Staubli VAL3: Rob6x.pjx

--- Rob6x.pjx ---
Parameters version=s7.9.1 stackSize=5000 millimeterUnit=true
Program file=AsynchStop.pgx
Program file=BytesToS16.pgx
Program file=Calibrate.pgx
Program file=CheckLimits.pgx
Program file=CheckStatus.pgx
Program file=Com.pgx
Program file=COM_SERIAL.pgx
Program file=Command.pgx
Program file=crc16.pgx
Program file=DeletePoint.pgx
Program file=Energize.pgx
Program file=FloatToBytes.pgx
Program file=GetAppVersion.pgx
Program file=GetCurrentPos.pgx
Program file=GetFirmVersion.pgx
Program file=GetJointPos.pgx
Program file=GetLimits.pgx
Program file=GetSerialNumber.pgx
Program file=GetSNCtrl.pgx
Program file=GetToolParam6x.pgx
Program file=GotoPoint.pgx
Program file=GotoPosition.pgx
Program file=Init.pgx
Program file=InitRobot.pgx
Program file=Input.pgx
Program file=isInLimits.pgx
Program file=KillAlltasks.pgx
Program file=MemPointPos.pgx
Program file=Motion.pgx
Program file=Move.pgx
Program file=MoveJoint.pgx
Program file=MoveJointTo.pgx
Program file=Output.pgx
Program file=SetAccel.pgx
Program file=SetLimits.pgx
Program file=SetSpeed.pgx
Program file=SetTool.pgx
Program file=SetToolParam.pgx
Program file=SetToolParam6x.pgx
Program file=start.pgx
Program file=stop.pgx
Program file=StopLimits.pgx
Program file=taskRecord.pgx
Program file=test.pgx
Program file=Valve.pgx
Data file=Rob6x.dtx

--- CheckLimits.pgx ---
program CheckLimits()
  local pointRx pt
  local bool curErr_Z
  local bool err_x
  local bool err_y
  local bool curErr_Y
  local bool err_z
  local num hysteresis
  local bool curErr_X
  local bool inLimits
  local num hysteresisZmin
begin
//*******************************************************************************
//*   ______
//*  / _____) /|
//* | |      / /
//* | | /\  / /
//* | | \ \/ /  _      Copyright (c) KEOLABS, 2016
//* | |  \__/  | |        http://www.keolabs.com
//* | |________| |
//*  \__________/
//*
//********************************************************************************
//*@file          : CheckLimits
//*@author        : Yves Ragot
//*@version       : $Id: CheckLimits.pgx 1645 2017-01-24 08:09:09Z yves $
//*@brief         : Check the if the current mouvement is in the limits
//*
//*******************************************************************************/

  // hysteresis in mm
  hysteresis = 70
  hysteresisZmin = 10

  do

      // get current position
      pt = here(tCurrentTool, fCurrentFrame)

      // round values before comparing with limits (integer values)
      pt.trsf.x = round(pt.trsf.x * 10) / 10
      pt.trsf.y = round(pt.trsf.y * 10) / 10
      pt.trsf.z = round(pt.trsf.z * 10) / 10

      // check first non fatal X limits
      if ((pt.trsf.x < CurLimitsTable["Xmin"]) or (pt.trsf.x > CurLimitsTable["Xmax"]))
          if (!curErr_X)
              call StopLimits()
          endIf
      else
          curErr_X = false
      endIf

      if ((pt.trsf.x >= CurLimitsTable["Xmin"] - hysteresis) and (pt.trsf.x <= CurLimitsTable["Xmax"] + hysteresis))
          curErr_X = true
      else
          call StopLimits()
      endIf

      // check first non fatal Y limits
      if ((pt.trsf.y < CurLimitsTable["Ymin"]) or (pt.trsf.y > CurLimitsTable["Ymax"]))
          if (!curErr_Y)
              call StopLimits()
          endIf
      else
          curErr_Y = false
      endIf

      if ((pt.trsf.y >= CurLimitsTable["Ymin"] - hysteresis) and (pt.trsf.y <= CurLimitsTable["Ymax"] + hysteresis))
          curErr_Y = true
      else
          call StopLimits()
      endIf

      // check first non fatal Z limits
      if ((pt.trsf.z < CurLimitsTable["Zmin"]) or (pt.trsf.z > CurLimitsTable["Zmax"]))
          if (!curErr_Z)
              call StopLimits()
          endIf
      else
          curErr_Z = false
      endIf

      if ((pt.trsf.z >= CurLimitsTable["Zmin"] - hysteresisZmin) and (pt.trsf.z <= CurLimitsTable["Zmax"] + hysteresis))
          curErr_Z = true
      else
          call StopLimits()
      endIf

     delay(0)

  until false

end

--- CheckStatus.pgx ---
program CheckStatus()
  local num esState
  local num status_err
  local num com_err
  local num limits_err
  local num motion_err
  local num newErrorCode
begin
//*******************************************************************************
//*   ______
//*  / _____) /|
//* | |      / /
//* | | /\  / /
//* | | \ \/ /  _      Copyright (c) KEOLABS, 2016
//* | |  \__/  | |        http://www.keolabs.com
//* | |________| |
//*  \__________/
//*
//********************************************************************************
//*@file          : CheckStatus
//*@author        : Yves Ragot
//*@version       : $Id: CheckStatus.pgx 1365 2016-11-18 16:00:54Z yves $
//*@brief         : Check robot status (busy, runing, error ?)
//*
//*******************************************************************************/

  do

      //== get task errors ==
      com_err = taskStatus("COM")
      limits_err = taskStatus("CheckLimits")
      status_err = taskStatus("CheckStatus")
      motion_err = taskStatus("Motion")

      // update LastErrorCode (taskStatus: 0 = suspended, 1 = running, -1 = dead
      if ((com_err != 0) and (com_err != 1))
          newErrorCode = com_err
      elseIf (motion_err > 1)
          newErrorCode = motion_err
      elseIf ((limits_err != 0) and (limits_err != 1))
          newErrorCode = limits_err
      elseIf ((status_err != 0) and (status_err != 1))
          newErrorCode = status_err
      else
          newErrorCode = 0
      endIf

      //== GeneralStatus
      // emergency stop ?
      esState = esStatus()
      if (esState != 0)
          call AsynchStop()
          GeneralStatus = 105
          LastErrorCode = 0

      // mouvement error ?
      elseIf (GeneralStatus == 0)

        switch (newErrorCode)

          // mouvement
          case 81, 150, 153, 154
            GeneralStatus = 100
          break

          // parameter
          case 70, 100, 101, 102, 103, 104, 160, 161, 165
            GeneralStatus = 101
          break

          // system
          case -1, 40, 41, 60, 61, 90, 125, 250
            GeneralStatus = 102
          break

          // soft
          case 10, 11, 20, 21, 29, 30, 31, 32, 80, 82, 105, 106, 122, 123, 124, 162, 163, 164
            GeneralStatus = 103
          break

          default
          break

        endSwitch

        if (newErrorCode != 0)
            LastErrorCode = newErrorCode
        endIf

    endIf

      // kill motion task if fault
    //    if ((GeneralStatus > 1) and (LastErrorCode != 0) and ((LastErrorCode == motion_err) or (LastErrorCode == 153)))
    if ((MoveRunning and (GeneralStatus > 1) and ((LastErrorCode == motion_err) or (LastErrorCode == 153))))
        call AsynchStop()
        setMutex(MotionTaskMutex)
        if taskStatus("Motion") != -1
            taskKill("Motion")
            wait(taskStatus("Motion") == -1)
            ExecuteMotion = false
        endIf
        MotionTaskMutex = false
    endIf

    // check movement running
    if (GeneralStatus == 1)
        // is mouvement always running ?
        if (isSettled() and isEmpty())
            GeneralStatus = 0
            MoveRunning = false
        endIf
    endIf

   delay(0)

  until false

end

--- Com.pgx ---
program COM()
  local num nbBuffer
  local num nbSent
  local num dataIn[50]
  local num dataOut[32]
  local num crc_l
  local num crc_h
  local num ret
  local num lenDataIn
  local num lenDataOut
  local num answer
  local string stringAnswer
  local num i
  local num j
  local num arrayAnswer[6]
  local num buffer[64]
  local num l_nIndex
  local num cpt
  local num nbBufTcp
  local num bufferTCP[64]
begin
//*******************************************************************************
//*   ______
//*  / _____) /|
//* | |      / /
//* | | /\  / /
//* | | \ \/ /  _      Copyright (c) KEOLABS, 2016
//* | |  \__/  | |        http://www.keolabs.com
//* | |________| |
//*  \__________/
//*
//********************************************************************************
//*@file          : COM
//*@author        : Yves Ragot
//*@version       : $Id: Com.pgx 1608 2017-01-13 10:03:43Z yves $
//*@brief         : PC socket communication management
//*
//*******************************************************************************/

  //== configuration socket ==
  // 1 seul client
  ret = sioCtrl(siTcpServer, "clients", 1)

  // timeout = 10ms
  ret = sioCtrl(siTcpServer, "timeout", 0.01)

  // buffers length
  lenDataIn = 32
  lenDataOut = 32

  NbCharReceived = 0
  ModeSerial = false

  // auto detection com port with first frame
  do
    nbBufTcp = sioGet(siTcpServer, bufferTCP)
  until ((NbBufSerial > 0) or (nbBufTcp > 0))

  // serial detection done by COM_SERIAL task
  if (NbBufSerial > 0)
      nbBuffer = NbBufSerial
      ModeSerial = true
  endIf
  if (nbBufTcp > 0)
      nbBuffer = nbBufTcp
      ModeSerial = false
  endIf

  if (nbBuffer > lenDataIn)
      nbBuffer = lenDataIn
  endIf

  if (ModeSerial)
      for l_nIndex = 0 to nbBuffer
          dataIn[NbCharReceived + l_nIndex] = BufferSerial[l_nIndex]
      endFor
  else
      for l_nIndex = 0 to nbBuffer
          dataIn[NbCharReceived + l_nIndex] = bufferTCP[l_nIndex]
      endFor
  endIf

  NbCharReceived = NbCharReceived + nbBuffer

  // main loop
  do

      cpt = 0

      do
          if (ModeSerial)
              nbBuffer = sioGet(siSerial1, buffer)
          else
              nbBuffer = sioGet(siTcpServer, buffer)
          endIf

          if (nbBuffer > 0)
              if (nbBuffer > lenDataIn)
                  nbBuffer = lenDataIn
              endIf
              if (NbCharReceived + nbBuffer > lenDataIn)
                  NbCharReceived = lenDataIn
              else

                  for l_nIndex = 0 to nbBuffer
                      dataIn[NbCharReceived + l_nIndex] = buffer[l_nIndex]
                  endFor
                  NbCharReceived = NbCharReceived + nbBuffer
                  cpt = cpt + 1
              endIf

          endIf

      // loop on charactere until all frame or 1s timeout
      until (NbCharReceived == lenDataIn) or cpt > 100

    if (NbCharReceived == lenDataIn)

      // check CRC
      call crc16(lenDataIn - 2, crc_h, crc_l, dataIn)

      if ((dataIn[lenDataIn - 2] != crc_h) or (dataIn[lenDataIn - 1] != crc_l))
          FrameReceiveNOK = FrameReceiveNOK + 1
      else
          FrameReceiveOK = FrameReceiveOK + 1

        //== command treatment ==
        setMutex(MotionTaskMutex)
        if  (taskStatus("Motion") == -1)
            taskCreate "Motion", 100, Motion()
        endIf

        // be sure that the task is running
        wait(taskStatus("Motion") == 1)
        MotionTaskMutex = false

        call Command(ret, dataIn, answer, stringAnswer, arrayAnswer)

        //== prepare response ==

        // command number
        dataOut[0] = dataIn[0]

        // frame number
        dataOut[1] = dataIn[1]

        // last error code
        dataOut[2] = LastErrorCode

        // status
        dataOut[3] = GeneralStatus

        // check response type
        switch (dataIn[0])

          // string
          case 10, 11, 13, 15
              for i = 0 to len(stringAnswer) - 1
                  dataOut[4 + i] = asc(stringAnswer, i)
              endFor
              for j = i to 24
                  dataOut[4 + j] = 0
              endFor
          break

          // numerical or nothing
          default
              // if not limits or ToolParam
              if ((dataIn[0] != 6) and (dataIn[0] != 16))
                  // current Cartesian position
                  call GetCurrentPos(arrayAnswer)
              endIf

              call FloatToBytes(arrayAnswer[0], dataOut[4], dataOut[5])
              call FloatToBytes(arrayAnswer[1], dataOut[6], dataOut[7])
              call FloatToBytes(arrayAnswer[2], dataOut[8], dataOut[9])
              call FloatToBytes(arrayAnswer[3], dataOut[10], dataOut[11])
              call FloatToBytes(arrayAnswer[4], dataOut[12], dataOut[13])
              call FloatToBytes(arrayAnswer[5], dataOut[14], dataOut[15])

              // current Joint position
              call GetJointPos(arrayAnswer)
              call FloatToBytes(arrayAnswer[0], dataOut[16], dataOut[17])
              call FloatToBytes(arrayAnswer[1], dataOut[18], dataOut[19])
              call FloatToBytes(arrayAnswer[2], dataOut[20], dataOut[21])
              call FloatToBytes(arrayAnswer[3], dataOut[22], dataOut[23])
              call FloatToBytes(arrayAnswer[4], dataOut[24], dataOut[25])
              call FloatToBytes(arrayAnswer[5], dataOut[26], dataOut[27])

              // command response (GetAccel/GetSpeed/GetToolParam or not)
              if (dataIn[0] == 3) or (dataIn[0] == 4) or (dataIn[0] == 5)
                  call FloatToBytes(answer, dataOut[28], dataOut[29])
              else
                  dataOut[28] = answer
              endIf
            break

        endSwitch

          // compute CRC
          call crc16(lenDataOut - 2, crc_h, crc_l, dataOut)
          dataOut[lenDataOut - 2] = crc_h
          dataOut[lenDataOut - 1] = crc_l

        // send response
        if (ModeSerial)
            nbSent = sioSet(siSerial1, dataOut)
        else
            nbSent = sioSet(siTcpServer, dataOut)
        endIf

        if (nbSent != lenDataOut)
            // TODO error
        endIf

        //if ((dataIn[30] != crc_h) or (dataIn[31] != crc_l))
      endIf

        //if (nbReceived == lenDataIn)
      elseIf (NbCharReceived > 0)
          FrameReceiveNOK = FrameReceiveNOK + 1
      endIf

      NbCharReceived = 0

      delay(0)

  until(bExit)

end

--- DeletePoint.pgx ---
program DeletePoint(num& bufferIn[])
  local string pointName
  local num i
begin
  //*******************************************************************************
  //*   ______
  //*  / _____) /|
  //* | |      / /
  //* | | /\  / /
  //* | | \ \/ /  _      Copyright (c) KEOLABS, 2016
  //* | |  \__/  | |        http://www.keolabs.com
  //* | |________| |
  //*  \__________/
  //*
  //********************************************************************************
  //*@file          : DeletePoint
  //*@author        : Yves Ragot
  //*@version       : $Id: DeletePoint.pgx 1198 2016-10-07 06:48:14Z yves $
  //*@brief         : Forget a memorized position point
  //*
  //*******************************************************************************/

  pointName = ""

  // get the name of the point
  for i = 0 to 9
      pointName = pointName + chr(bufferIn[17 + i])
  endFor

  if (len(pointName)) > 0

      // delete the point from the collection
      if (isDefined(pPointsTable[pointName]) == true)
          delete(pPointsTable[pointName])
      else
          GeneralStatus = 101
          LastErrorCode = 0
      endIf

  else
      GeneralStatus = 101
      LastErrorCode = 0
  endIf

end

--- GetAppVersion.pgx ---
program GetAppVersion(string& answer)
begin
//*******************************************************************************
//*   ______
//*  / _____) /|
//* | |      / /
//* | | /\  / /
//* | | \ \/ /  _      Copyright (c) KEOLABS, 2016
//* | |  \__/  | |        http://www.keolabs.com
//* | |________| |
//*  \__________/
//*
//********************************************************************************
//*@file          : GetAppVersion
//*@author        : Yves Ragot
//*@version       : $Id: GetAppVersion.pgx 1645 2017-01-24 08:09:09Z yves $
//*@brief         : Get firmware version (application version)
//*******************************************************************************/

  answer = "v1.1 jan 23 2017"

end

--- GetJointPos.pgx ---
program GetJointPos(num& posArray[])
  local jointRx jt
begin
  //*******************************************************************************
  //*   ______
  //*  / _____) /|
  //* | |      / /
  //* | | /\  / /
  //* | | \ \/ /  _      Copyright (c) KEOLABS, 2016
  //* | |  \__/  | |        http://www.keolabs.com
  //* | |________| |
  //*  \__________/
  //*
  //********************************************************************************
  //*@file          : GetJointPos
  //*@author        : Yves Ragot
  //*@version       : $Id: GetJointPos.pgx 1198 2016-10-07 06:48:14Z yves $
  //*@brief         : Get current joint position
  //*
  //*******************************************************************************/

  // get joint position and converts to 1/10 mm
  jt = herej()
  posArray[0] = jt.j1 * 10
  posArray[1] = jt.j2 * 10
  posArray[2] = jt.j3 * 10
  posArray[3] = jt.j4 * 10
  posArray[4] = jt.j5 * 10
  posArray[5] = jt.j6 * 10

end

--- GetLimits.pgx ---
program GetLimits(num& limits[])
begin
  //*******************************************************************************
  //*   ______
  //*  / _____) /|
  //* | |      / /
  //* | | /\  / /
  //* | | \ \/ /  _      Copyright (c) KEOLABS, 2016
  //* | |  \__/  | |        http://www.keolabs.com
  //* | |________| |
  //*  \__________/
  //*
  //********************************************************************************
  //*@file          : GetLimits
  //*@author        : Yves Ragot
  //*@version       : $Id: GetLimits.pgx 1198 2016-10-07 06:48:14Z yves $
  //*@brief         : Get limits
  //*
  //*******************************************************************************/

  // get limits table elements and converts to 1/10 mm
  limits[0] = CurLimitsTable["Xmin"] * 10
  limits[1] = CurLimitsTable["Ymin"] * 10
  limits[2] = CurLimitsTable["Zmin"] * 10
  limits[3] = CurLimitsTable["Xmax"] * 10
  limits[4] = CurLimitsTable["Ymax"] * 10
  limits[5] = CurLimitsTable["Zmax"] * 10

end

--- GetSNCtrl.pgx ---
program GetSNCtrl(string answer)
begin
//*******************************************************************************
//*   ______
//*  / _____) /|
//* | |      / /
//* | | /\  / /
//* | | \ \/ /  _      Copyright (c) KEOLABS, 2016
//* | |  \__/  | |        http://www.keolabs.com
//* | |________| |
//*  \__________/
//*
//********************************************************************************
//*@file          : GetSNCtrl
//*@author        : Yves Ragot
//*@version       : $Id: GetSNCtrl.pgx 1193 2016-10-06 09:55:11Z yves $
//*@brief         : Get Serial Number of the controller
//*
//*******************************************************************************/

  answer = left(getVersion("ControllerSN"), 20)

end

--- GotoPoint.pgx ---
program GotoPoint(num& bufferIn[])
  local string pointName
  local num i
begin
//*******************************************************************************
//*   ______
//*  / _____) /|
//* | |      / /
//* | | /\  / /
//* | | \ \/ /  _      Copyright (c) KEOLABS, 2016
//* | |  \__/  | |        http://www.keolabs.com
//* | |________| |
//*  \__________/
//*
//********************************************************************************
//*@file          : GotoPoint
//*@author        : Yves Ragot
//*@version       : $Id: GotoPoint.pgx 1291 2016-10-25 14:40:00Z yves $
//*@brief         : Go to a memorized point
//*
//*******************************************************************************/

  pointName = ""

  // get the name of the point
  for i = 0 to 9
      pointName = pointName + chr(bufferIn[17 + i])
  endFor

  if (len(pointName)) > 0

      // is the point previously defined in the collection
      if (isDefined(pPointsTable[pointName]) == true)

          pTargetPoint = pPointsTable[pointName]

          CartesianMode = true

          // launch mouvement
          ExecuteMotion = true

          // wait for end of execution
          wait(ExecuteMotion == false)

      else
          GeneralStatus = 101
          LastErrorCode = 0
      endIf

  else
      GeneralStatus = 101
      LastErrorCode = 0
  endIf

end

--- Init.pgx ---
program Init()
begin
//*******************************************************************************
//*   ______
//*  / _____) /|
//* | |      / /
//* | | /\  / /
//* | | \ \/ /  _      Copyright (c) KEOLABS, 2016
//* | |  \__/  | |        http://www.keolabs.com
//* | |________| |
//*  \__________/
//*
//********************************************************************************
//*@file          : Init
//*@author        : Yves Ragot
//*@version       : $Id: Init.pgx 1645 2017-01-24 08:09:09Z yves $
//*@brief         : global program initialization
//*
//*******************************************************************************/

  // creation limits table with default values
  insert(CurLimitsTable["Xmin"])
  CurLimitsTable["Xmin"] = -310
  insert(CurLimitsTable["Xmax"])
  CurLimitsTable["Xmax"] = 545
  insert(CurLimitsTable["Ymin"])
  CurLimitsTable["Ymin"] = -210
  insert(CurLimitsTable["Ymax"])
  CurLimitsTable["Ymax"] = 210
  insert(CurLimitsTable["Zmin"])
  CurLimitsTable["Zmin"] = -310
  insert(CurLimitsTable["Zmax"])
  CurLimitsTable["Zmax"] = 520

// for test
//   insert(CurLimitsTable["Xmin"])
//  CurLimitsTable["Xmin"] = -1000
//  insert(CurLimitsTable["Xmax"])
//  CurLimitsTable["Xmax"] = 1000
//  insert(CurLimitsTable["Ymin"])
//  CurLimitsTable["Ymin"] = -1000
//  insert(CurLimitsTable["Ymax"])
//  CurLimitsTable["Ymax"] = 1000
//  insert(CurLimitsTable["Zmin"])
//  CurLimitsTable["Zmin"] = -1000
//  insert(CurLimitsTable["Zmax"])
//  CurLimitsTable["Zmax"] = 1000

  // Global varaibles initialization
  bExit = false
  CartesianMode = true
  AlignMode = false
  AsyncMode = true
  //tCurrentTool = flange
  //currentToolType = 99
  call SetToolParam(0)
  fCurrentFrame = world
  LastErrorCode = 0
  GeneralStatus = 0
  MoveRunning = false
  bStartRecording = false

  // Default accleration and speed
  COEFF_ACCEL = 3
  mNomSpeed.vel = 20
  mNomSpeed.accel = 50
  mNomSpeed.decel = 50

end

--- InitRobot.pgx ---
program InitRobot()
  local num maxSpeed
  local num cpt
begin
//*******************************************************************************
//*   ______
//*  / _____) /|
//* | |      / /
//* | | /\  / /
//* | | \ \/ /  _      Copyright (c) KEOLABS, 2016
//* | |  \__/  | |        http://www.keolabs.com
//* | |________| |
//*  \__________/
//*
//********************************************************************************
//*@file          : InitRobot
//*@author        : Yves Ragot
//*@version       : $Id: InitRobot.pgx 1658 2017-01-25 07:36:52Z yves $
//*@brief         : InitRobot command treatment
//*
//*******************************************************************************/

  // reinit default values
  call Init()

  // remote ?
  if (workingMode() != 4)
      popUpMsg("Please switch to remote mode")
      GeneralStatus = 106
  else
      // auto connection mouvement in remote mode
      autoConnectMove(true)

      // reset motion task
      resetMotion()

      // power
      enablePower()
      cpt = 0
      do
        delay(0.1)
        cpt = cpt + 1
      until (isPowered() or (cpt >  50))

      if (cpt > 50)
          GeneralStatus = 106
      else
          //set max speed
          maxSpeed = getMonitorSpeed()
          if (maxSpeed < 100)
              setMonitorSpeed(100)
          endIf
      endIf
  endIf
end

--- isInLimits.pgx ---
program IsInLimits(bool& ret)
  local pointRx pt
  local bool err_x
  local bool err_y
  local bool err_z
begin
//*******************************************************************************
//*   ______
//*  / _____) /|
//* | |      / /
//* | | /\  / /
//* | | \ \/ /  _      Copyright (c) KEOLABS, 2016
//* | |  \__/  | |        http://www.keolabs.com
//* | |________| |
//*  \__________/
//*
//********************************************************************************
//*@file          : IsInLimits
//*@author        : Yves Ragot
//*@version       : $Id: isInLimits.pgx 1558 2017-01-05 08:13:36Z yves $
//*@brief         : Check the if the current position is in the limits
//*
//*******************************************************************************/

  // get current position
  pt = here(tCurrentTool, fCurrentFrame)

  // round values before comparing with limits (integer values)
  pt.trsf.x = round(pt.trsf.x * 10) / 10
  pt.trsf.y = round(pt.trsf.y * 10) / 10
  pt.trsf.z = round(pt.trsf.z * 10) / 10

  // check fatal limits
  err_x = (pt.trsf.x < CurLimitsTable["Xmin"]) or (pt.trsf.x > CurLimitsTable["Xmax"])
  err_y = (pt.trsf.y < CurLimitsTable["Ymin"]) or (pt.trsf.y > CurLimitsTable["Ymax"])
  err_z = (pt.trsf.z < CurLimitsTable["Zmin"]) or (pt.trsf.z > CurLimitsTable["Zmax"])

  // ret = true if position is correctly in limits
  ret = !(err_x or err_y or err_z)

end

--- MemPointPos.pgx ---
program MemPointPos(num& bufferIn[])
  local string pointName
  local num i
  local pointRx pt
  local num result
begin
  //*******************************************************************************
  //*   ______
  //*  / _____) /|
  //* | |      / /
  //* | | /\  / /
  //* | | \ \/ /  _      Copyright (c) KEOLABS, 2016
  //* | |  \__/  | |        http://www.keolabs.com
  //* | |________| |
  //*  \__________/
  //*
  //********************************************************************************
  //*@file          : MemPointPos
  //*@author        : Yves Ragot
  //*@version       : $Id: MemPointPos.pgx 1291 2016-10-25 14:40:00Z yves $
  //*@brief         : Memorization of position point
  //*
  //*******************************************************************************/

  pointName = ""

  // get the name of the point
  for i = 0 to 9
      pointName = pointName + chr(bufferIn[17 + i])
  endFor

  if (len(pointName)) > 0

      // get position of the point
      call BytesToS16(bufferIn[3], bufferIn[4], result)
      pt.trsf.x = result / 10

      call BytesToS16(bufferIn[5], bufferIn[6], result)
      pt.trsf.y = result / 10

      call BytesToS16(bufferIn[7], bufferIn[8], result)
      pt.trsf.z = result / 10

      call BytesToS16(bufferIn[9], bufferIn[10], result)
      pt.trsf.rx = result / 10

      call BytesToS16(bufferIn[11], bufferIn[12], result)
      pt.trsf.ry = result / 10

      call BytesToS16(bufferIn[13], bufferIn[14], result)
      pt.trsf.rz = result / 10

      link(pt, fCurrentFrame)

      // insert the point into the collection
      if (isDefined(pPointsTable[pointName]) == false)
          insert(pPointsTable[pointName])
          pPointsTable[pointName] = pt
      else
          GeneralStatus = 101
          LastErrorCode = 0
      endIf

  else
    GeneralStatus = 101
    LastErrorCode = 0
  endIf

end

--- Move.pgx ---
program Move(num& arrayValue[])
  local pointRx pt
begin
//*******************************************************************************
//*   ______
//*  / _____) /|
//* | |      / /
//* | | /\  / /
//* | | \ \/ /  _      Copyright (c) KEOLABS, 2016
//* | |  \__/  | |        http://www.keolabs.com
//* | |________| |
//*  \__________/
//*
//********************************************************************************
//*@file          : Move
//*@author        : Yves Ragot
//*@version       : $Id: Move.pgx 1198 2016-10-07 06:48:14Z yves $
//*@brief         : Move command treatment (relative mouvement)
//*
//*******************************************************************************/

  // current Cartesian position
  pt = here(tCurrentTool, fCurrentFrame)

  // get and compute target point
  pTargetPoint.trsf.x = pt.trsf.x + arrayValue[0]
  pTargetPoint.trsf.y = pt.trsf.y + arrayValue[1]
  pTargetPoint.trsf.z = pt.trsf.z + arrayValue[2]
  pTargetPoint.trsf.rx = pt.trsf.rx + arrayValue[3]
  pTargetPoint.trsf.ry = pt.trsf.ry + arrayValue[4]
  pTargetPoint.trsf.rz = pt.trsf.rz + arrayValue[5]

  CartesianMode = true

  // launch mouvement
  ExecuteMotion = true

  // wait for end of execution
  wait(ExecuteMotion == false)

end

--- SetSpeed.pgx ---
program SetSpeed(num value)
begin
  //*******************************************************************************
  //*   ______
  //*  / _____) /|
  //* | |      / /
  //* | | /\  / /
  //* | | \ \/ /  _      Copyright (c) KEOLABS, 2016
  //* | |  \__/  | |        http://www.keolabs.com
  //* | |________| |
  //*  \__________/
  //*
  //********************************************************************************
  //*@file          : SetSpeed
  //*@author        : Yves Ragot
  //*@version       : $Id: SetSpeed.pgx 1644 2017-01-24 08:08:07Z yves $
  //*@brief         : Change speed parameter
  //*
  //*******************************************************************************/

  if ((value > 0) and (value <= 10000))

      // max translation speed
      mNomSpeed.tvel = value

      // max rotation speed
      mNomSpeed.vel = value / 10
      if (mNomSpeed.vel) > 100
          mNomSpeed.vel = 100
      endIf
  else
      GeneralStatus = 101
      LastErrorCode = 0
  endIf

end

--- SetToolParam.pgx ---
program SetToolParam(num value)
  local num prevType
  local tool prevTool
  local bool inLimits
begin
  //*******************************************************************************
  //*   ______
  //*  / _____) /|
  //* | |      / /
  //* | | /\  / /
  //* | | \ \/ /  _      Copyright (c) KEOLABS, 2016
  //* | |  \__/  | |        http://www.keolabs.com
  //* | |________| |
  //*  \__________/
  //*
  //********************************************************************************
  //*@file          : SetToolParam
  //*@author        : Yves Ragot
  //*@version       : $Id: SetToolParam.pgx 1490 2016-12-14 15:39:12Z yves $
  //*@brief         : Set the length of the tool
  //*
  //*******************************************************************************/

  // save previous tool parameter
  prevTool = tCurrentTool
  prevType = currentToolType

  // set new tool
  tCurrentTool = flange
  tCurrentTool.trsf.z = value
  tCurrentTool.trsf.rx = -180
  tCurrentTool.trsf.rz = 180
  currentToolType = 99

  // check if current position with new tool is in new limits
  call IsInLimits(inLimits)

  // if not, error
  if (!inLimits)

      // restore previous limits
      tCurrentTool = prevTool
      currentToolType = prevType

      // parameter error
      GeneralStatus = 101
      LastErrorCode = 0

  endIf

end

--- test.pgx ---
program test()
  local num lenDataOut
  local joint j
  local pointRx pt
  local num ret
  local num crc_h
  local num crc_l
  local num lenDataIn
  local num l_nNum
  local num dataOut[32]
  local num nbReceived
  local num nbSent
  local num dataIn[50]
  local num cycleCount
begin
//*******************************************************************************
//*   ______
//*  / _____) /|
//* | |      / /
//* | | /\  / /
//* | | \ \/ /  _      Copyright (c) KEOLABS, 2016
//* | |  \__/  | |        http://www.keolabs.com
//* | |________| |
//*  \__________/
//*
//********************************************************************************
//*@file          : test
//*@author        : Yves Ragot
//*@version       : $Id: test.pgx 1267 2016-10-17 13:45:02Z yves $
//*@brief         : PC socket communication simulation for test
//*
//*******************************************************************************/

  //== configuration socket ==
  // IP PC
  //ret = sioCtrl(siTcpClient, "target", "192.168.30.118")

  // no timeout
  ret = sioCtrl(siTcpClient, "timeout", 0)

  // buffers length
  lenDataIn = 32
  lenDataOut = 32

  cycleCount = 0

  do
      //== prepare resquest ==
      if (cycleCount == 0)
          dataOut[0] = 1
      else
          dataOut[0] = 101
      endIf

      // frame number
      dataOut[1] = dataOut[1] + 1

      // RFU
      dataOut[2] = 0

      // target Cartesian position
       //pt = here(tCurrentTool, fCurrentFrame)
      if ((cycleCount % 2) != 0)
          pt.trsf = {2000, 2000, -1000, 0, 0, 0}
      else
          pt.trsf = {-2000, 2000, -2000, 0, 0, 0}
      endIf

      dataOut[3] = roundDown(pt.trsf.x / 256)
      dataOut[4] =  bAnd(pt.trsf.x, 255)
      dataOut[5] = roundDown(pt.trsf.y / 256)
      dataOut[6] =  bAnd(pt.trsf.y, 255)
      dataOut[7] = roundDown(pt.trsf.z / 256)
      dataOut[8] =  bAnd(pt.trsf.z, 255)
      dataOut[9] = roundDown(pt.trsf.rx / 256)
      dataOut[10] =  bAnd(pt.trsf.rx, 255)
      dataOut[11] = roundDown(pt.trsf.ry / 256)
      dataOut[12] =  bAnd(pt.trsf.ry, 255)
      dataOut[13] = roundDown(pt.trsf.rz / 256)
      dataOut[14] =  bAnd(pt.trsf.rz, 255)

      // target Joint position
      //j = herej()
//      dataOut[3]  = roundDown(j.j1 / 256)
//      dataOut[4]  =  bAnd(j.j1, 255)
//      dataOut[5]  = roundDown(j.j2 / 256)
//      dataOut[6]  =  bAnd(j.j2, 255)
//      dataOut[7]  = roundDown(j.j3 / 256)
//      dataOut[8]  =  bAnd(j.j3, 255)
//      dataOut[9]  = roundDown(j.j4 / 256)
//      dataOut[10] =  bAnd(j.j4, 255)
//      dataOut[11] = roundDown(j.j5 / 256)
//      dataOut[12] =  bAnd(j.j5, 255)
//      dataOut[13] = roundDown(j.j6 / 256)
//      dataOut[14] =  bAnd(j.j6, 255)

      // RFU
      dataOut[15] = 0

      // asynchronous mode ?
      dataOut[16] = 0

      // point name
      dataOut[17] = 0
      dataOut[18] = 0
      dataOut[19] = 0
      dataOut[20] = 0
      dataOut[21] = 0
      dataOut[22] = 0
      dataOut[23] = 0
      dataOut[24] = 0
      dataOut[25] = 0
      dataOut[26] = 0

      // RFU
      dataOut[27] = 0
      dataOut[28] = 0
      dataOut[29] = 0

      // compute CRC
      call crc16(lenDataOut - 2, crc_h, crc_l, dataOut)
      dataOut[30] = crc_h
      dataOut[31] = crc_l

      // send response
      nbSent = sioSet(siTcpClient, dataOut)
      if (nbSent != lenDataOut)
          // TODO error
          put(nbSent)
      endIf

        //if ((dataIn[30] != crc_h) or (dataIn[31] != crc_l))

      nbReceived = sioGet(siTcpClient, dataIn)
      if (nbReceived == lenDataIn)

          // check CRC
          call crc16(lenDataIn - 2, crc_h, crc_l, dataIn)

          if ((dataIn[30] != crc_h) or (dataIn[31] != crc_l))
              FrameReceiveNOK = FrameReceiveNOK + 1
          else
              FrameReceiveOK = FrameReceiveOK + 1
          endIf

      //if (nbReceived == lenDataIn)
      else
          FrameReceiveNOK = FrameReceiveNOK + 1
      endIf

      cycleCount = cycleCount + 1
      delay(1)

  until(bExit)

end

--- Valve.pgx ---
program Valve(bool cde)
begin
  //*******************************************************************************
  //*   ______
  //*  / _____) /|
  //* | |      / /
  //* | | /\  / /
  //* | | \ \/ /  _      Copyright (c) KEOLABS, 2016
  //* | |  \__/  | |        http://www.keolabs.com
  //* | |________| |
  //*  \__________/
  //*
  //********************************************************************************
  //*@file          : Valve
  //*@author        : Yves Ragot
  //*@version       : $Id: Valve.pgx 1882 2019-01-10 16:18:45Z xavier $
  //*@brief         : Valve command
  //*
  //*******************************************************************************/

  //valve1 = cde
  if (cde)
    open(tCurrentTool)
  else
    close(tCurrentTool)
  endIf

end
